(*

.. <legal notes>

legal notes
=================
| SPDX-FileCopyrightText: © 2026 Oleksandr Tiutyk <trofimich@gmail.com>
| SPDX-License-Identifier: LGPL-3.0-only
| For details check: LGPL-3.0-only_

.. _LGPL-3.0-only: https://www.gnu.org/licenses/lgpl-3.0.en.html

.. </legal notes>

*)

{attribute 'qualified_only'}
{attribute 'strict'}
{attribute 'to_string'}
TYPE AUTOMATION_CONTROLLER_STATE :
(
	INITIAL := 0,
    WORKING := 1,            
    FAULT := 2
);
END_TYPE

(* stored: Version 1.1.0.1
   DUT AUTOMATION_CONTROLLER_STATE: Id {3a7a0191-f562-4dbc-a295-c4fdddac5490} *)
